// TIA Portal V16 export
// export: Created 2023-03-29T11:04:38.4378886Z, ExportSetting WithDefaults, DisplayName Totally Integrated Automation Portal, DisplayVersion V16 Update 6, DisplayName TIA Portal Version Control Interface, DisplayVersion V16 Update 2, DisplayName TIA Portal Openness, DisplayVersion V16 Update 6, DisplayName STEP 7 Professional, DisplayVersion V16 Update 6, DisplayName STEP 7 Safety, DisplayVersion V16, DisplayName WinCC Advanced, DisplayVersion V16 Update 6
FUNCTION "MPP04_2_rez" : Void   // FC24, LAD
TITLE = Read data from SC100
{ S7_Optimized_Access := 'TRUE' }
AUTHOR : rtecmer
VERSION : 0.1
// Czytanie z SC1000 
// Obsługa protokołu Master Modbus RTU.  Odczyt pomiarów  i status czujnika SC1000
// stored: AutoNumber false, IsIECCheckEnabled false, SetENOAutomatically false, UDAEnableTagReadback false
   VAR_TEMP
      Wielkość_przeływu_Adres0_0 : DWord;
      Wielkość_przeływu_Adres0_1 : DWord;
      Wielkość_przeływu_Adres2_0 : DWord;
      Wielkość_przeływu_Adres2_2 : DWord;
   END_VAR
   VAR_TEMP   // added for the SCL form of the ladder/FBD networks
      _w1 : Bool;
      _w2 : Bool;
   END_VAR
BEGIN

REGION Network 1
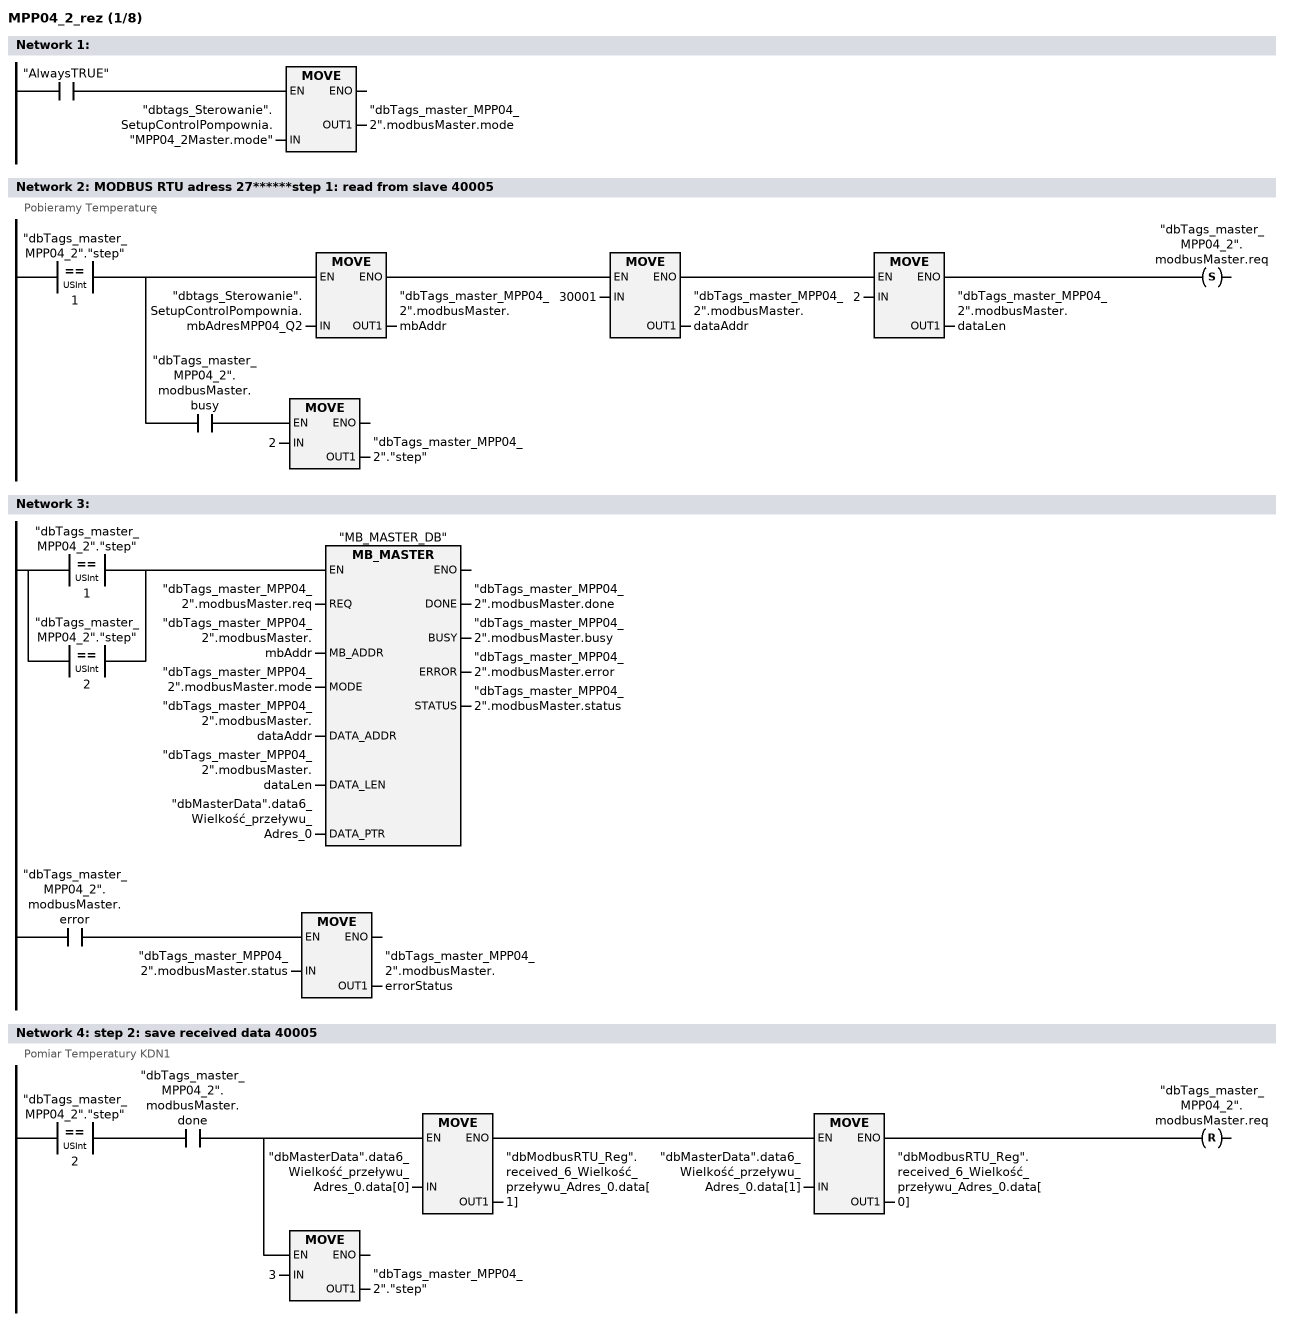
   RUNG wire#powerrail
      Contact( "AlwaysTRUE" )
      { S7_GenerateENO := "TRUE" } Move(in := "dbtags_Sterowanie".SetupControlPompownia."MPP04_2Master.mode", out1 => "dbTags_master_MPP04_2".modbusMaster.mode)
   END_RUNG
   // the same network as SCL:
   IF "AlwaysTRUE" THEN
       "dbTags_master_MPP04_2".modbusMaster.mode := "dbtags_Sterowanie".SetupControlPompownia."MPP04_2Master.mode";
   END_IF;
END_REGION

REGION Network 2: MODBUS RTU adress 27******step 1: read from slave 40005
   // Pobieramy Temperaturę
   RUNG wire#powerrail
      { S7_Templates := "SrcType := USInt" } EQ_Contact(in1 := "dbTags_master_MPP04_2"."step", in2 := 1)
      wire#w1
      Move(in := "dbtags_Sterowanie".SetupControlPompownia.mbAdresMPP04_Q2, out1 => "dbTags_master_MPP04_2".modbusMaster.mbAddr)
      { S7_GenerateENO := "TRUE" } Move(in := 30001, out1 => "dbTags_master_MPP04_2".modbusMaster.dataAddr)
      Move(in := 2, out1 => "dbTags_master_MPP04_2".modbusMaster.dataLen)
      S_Coil( "dbTags_master_MPP04_2".modbusMaster.req )
   END_RUNG
   RUNG wire#w1
      Contact( "dbTags_master_MPP04_2".modbusMaster.busy )
      { S7_GenerateENO := "TRUE" } Move(in := 2, out1 => "dbTags_master_MPP04_2"."step")
   END_RUNG
   // the same network as SCL:
   // ENO of a box is taken as its EN; it also drops when the box reports an error
   #_w1 := "dbTags_master_MPP04_2"."step" = 1;
   IF #_w1 THEN
       "dbTags_master_MPP04_2".modbusMaster.mbAddr := "dbtags_Sterowanie".SetupControlPompownia.mbAdresMPP04_Q2;
       "dbTags_master_MPP04_2".modbusMaster.dataAddr := 30001;
       "dbTags_master_MPP04_2".modbusMaster.dataLen := 2;
       "dbTags_master_MPP04_2".modbusMaster.req := TRUE;
   END_IF;
   IF #_w1 AND "dbTags_master_MPP04_2".modbusMaster.busy THEN "dbTags_master_MPP04_2"."step" := 2; END_IF;
END_REGION

REGION Network 3
   RUNG wire#powerrail
      { S7_Templates := "SrcType := USInt" } EQ_Contact(in1 := "dbTags_master_MPP04_2"."step", in2 := 1)
      wire#w1
      "MB_MASTER_DB".MB_MASTER(REQ := "dbTags_master_MPP04_2".modbusMaster.req, MB_ADDR := "dbTags_master_MPP04_2".modbusMaster.mbAddr, MODE := "dbTags_master_MPP04_2".modbusMaster.mode, DATA_ADDR := "dbTags_master_MPP04_2".modbusMaster.dataAddr, DATA_LEN := "dbTags_master_MPP04_2".modbusMaster.dataLen, DATA_PTR := "dbMasterData".data6_Wielkość_przeływu_Adres_0, DONE => "dbTags_master_MPP04_2".modbusMaster.done, BUSY => "dbTags_master_MPP04_2".modbusMaster.busy, ERROR => "dbTags_master_MPP04_2".modbusMaster.error, STATUS => "dbTags_master_MPP04_2".modbusMaster.status)
   END_RUNG
   RUNG wire#powerrail
      { S7_Templates := "SrcType := USInt" } EQ_Contact(in1 := "dbTags_master_MPP04_2"."step", in2 := 2)
   END_RUNG wire#w1
   RUNG wire#powerrail
      Contact( "dbTags_master_MPP04_2".modbusMaster.error )
      { S7_GenerateENO := "TRUE" } Move(in := "dbTags_master_MPP04_2".modbusMaster.status, out1 => "dbTags_master_MPP04_2".modbusMaster.errorStatus)
   END_RUNG
   // the same network as SCL:
   IF ("dbTags_master_MPP04_2"."step" = 1) OR ("dbTags_master_MPP04_2"."step" = 2) THEN
       "MB_MASTER_DB"(REQ := "dbTags_master_MPP04_2".modbusMaster.req,   // MB_MASTER
                      MB_ADDR := "dbTags_master_MPP04_2".modbusMaster.mbAddr,
                      MODE := "dbTags_master_MPP04_2".modbusMaster.mode,
                      DATA_ADDR := "dbTags_master_MPP04_2".modbusMaster.dataAddr,
                      DATA_LEN := "dbTags_master_MPP04_2".modbusMaster.dataLen,
                      DATA_PTR := "dbMasterData".data6_Wielkość_przeływu_Adres_0,
                      DONE => "dbTags_master_MPP04_2".modbusMaster.done,
                      BUSY => "dbTags_master_MPP04_2".modbusMaster.busy,
                      ERROR => "dbTags_master_MPP04_2".modbusMaster.error,
                      STATUS => "dbTags_master_MPP04_2".modbusMaster.status);
   END_IF;
   IF "dbTags_master_MPP04_2".modbusMaster.error THEN
       "dbTags_master_MPP04_2".modbusMaster.errorStatus := "dbTags_master_MPP04_2".modbusMaster.status;
   END_IF;
END_REGION

REGION Network 4: step 2: save received data 40005
   // Pomiar Temperatury KDN1
   RUNG wire#powerrail
      { S7_Templates := "SrcType := USInt" } EQ_Contact(in1 := "dbTags_master_MPP04_2"."step", in2 := 2)
      Contact( "dbTags_master_MPP04_2".modbusMaster.done )
      wire#w1
      { S7_GenerateENO := "TRUE" } Move(in := "dbMasterData".data6_Wielkość_przeływu_Adres_0.data[0], out1 => "dbModbusRTU_Reg".received_6_Wielkość_przeływu_Adres_0.data[1])
      { S7_GenerateENO := "TRUE" } Move(in := "dbMasterData".data6_Wielkość_przeływu_Adres_0.data[1], out1 => "dbModbusRTU_Reg".received_6_Wielkość_przeływu_Adres_0.data[0])
      R_Coil( "dbTags_master_MPP04_2".modbusMaster.req )
   END_RUNG
   RUNG wire#w1
      { S7_GenerateENO := "TRUE" } Move(in := 3, out1 => "dbTags_master_MPP04_2"."step")
   END_RUNG
   // the same network as SCL:
   // ENO of a box is taken as its EN; it also drops when the box reports an error
   IF ("dbTags_master_MPP04_2"."step" = 2) AND "dbTags_master_MPP04_2".modbusMaster.done THEN
       "dbModbusRTU_Reg".received_6_Wielkość_przeływu_Adres_0.data[1] := "dbMasterData".data6_Wielkość_przeływu_Adres_0.data[0];
       "dbModbusRTU_Reg".received_6_Wielkość_przeływu_Adres_0.data[0] := "dbMasterData".data6_Wielkość_przeływu_Adres_0.data[1];
       "dbTags_master_MPP04_2".modbusMaster.req := FALSE;
       "dbTags_master_MPP04_2"."step" := 3;
   END_IF;
END_REGION

REGION Network 5: MODBUS RTU adress 27******step 3: read from slave 40001
   // Bytes Error
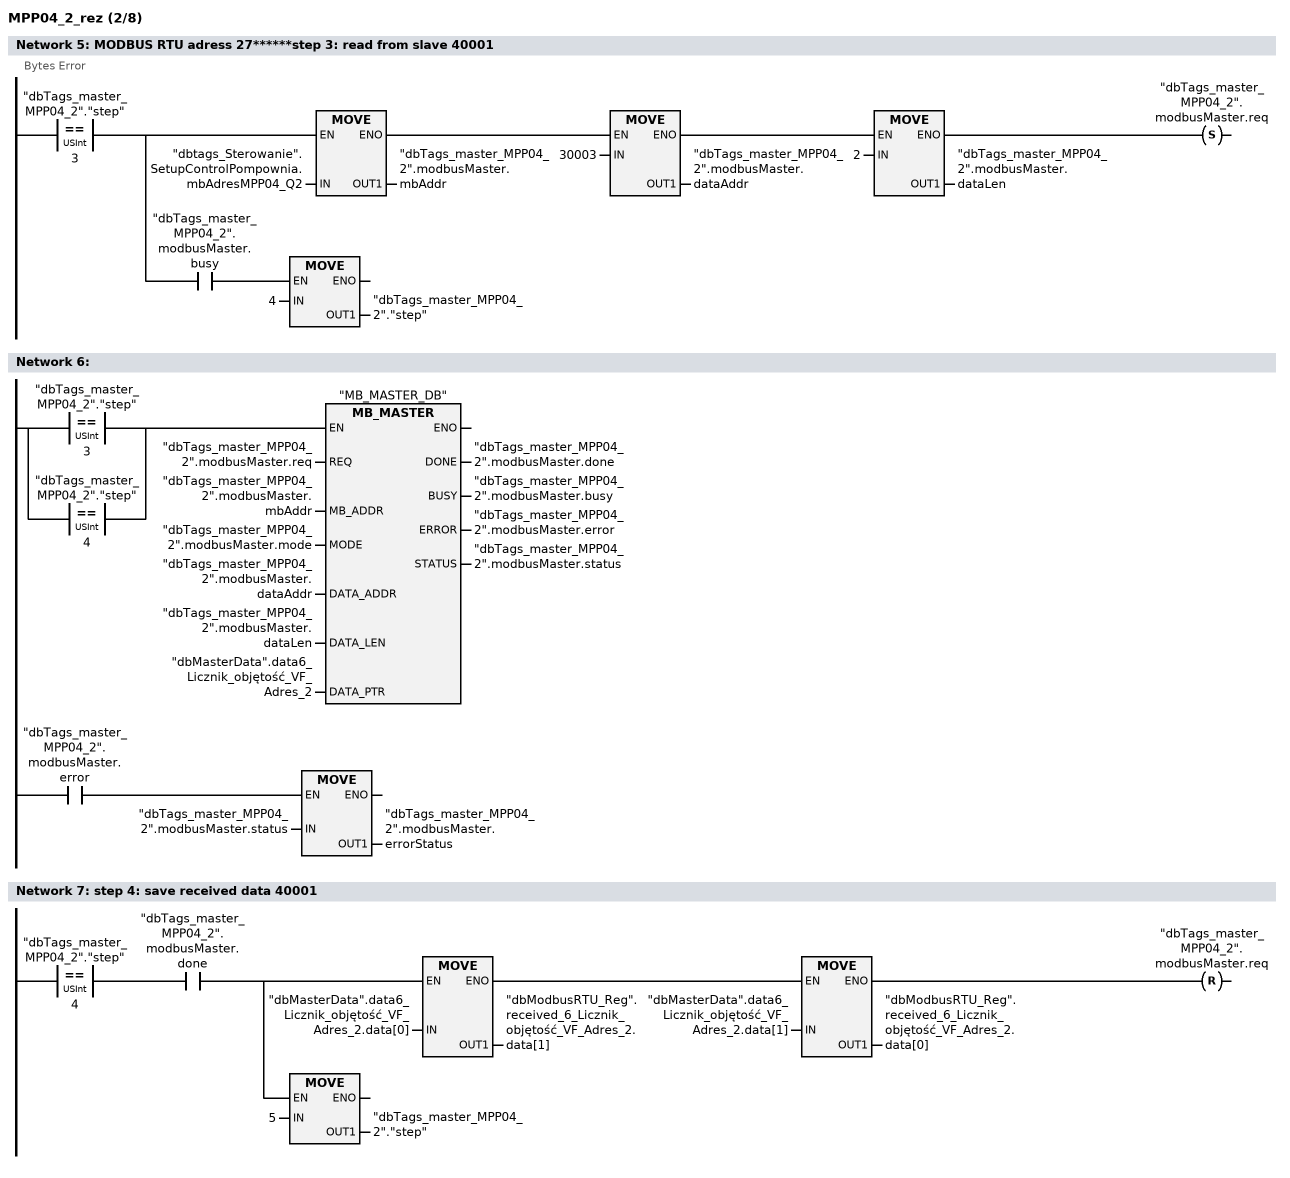
   RUNG wire#powerrail
      { S7_Templates := "SrcType := USInt" } EQ_Contact(in1 := "dbTags_master_MPP04_2"."step", in2 := 3)
      wire#w1
      Move(in := "dbtags_Sterowanie".SetupControlPompownia.mbAdresMPP04_Q2, out1 => "dbTags_master_MPP04_2".modbusMaster.mbAddr)
      { S7_GenerateENO := "TRUE" } Move(in := 30003, out1 => "dbTags_master_MPP04_2".modbusMaster.dataAddr)
      Move(in := 2, out1 => "dbTags_master_MPP04_2".modbusMaster.dataLen)
      S_Coil( "dbTags_master_MPP04_2".modbusMaster.req )
   END_RUNG
   RUNG wire#w1
      Contact( "dbTags_master_MPP04_2".modbusMaster.busy )
      { S7_GenerateENO := "TRUE" } Move(in := 4, out1 => "dbTags_master_MPP04_2"."step")
   END_RUNG
   // the same network as SCL:
   // ENO of a box is taken as its EN; it also drops when the box reports an error
   #_w1 := "dbTags_master_MPP04_2"."step" = 3;
   IF #_w1 THEN
       "dbTags_master_MPP04_2".modbusMaster.mbAddr := "dbtags_Sterowanie".SetupControlPompownia.mbAdresMPP04_Q2;
       "dbTags_master_MPP04_2".modbusMaster.dataAddr := 30003;
       "dbTags_master_MPP04_2".modbusMaster.dataLen := 2;
       "dbTags_master_MPP04_2".modbusMaster.req := TRUE;
   END_IF;
   IF #_w1 AND "dbTags_master_MPP04_2".modbusMaster.busy THEN "dbTags_master_MPP04_2"."step" := 4; END_IF;
END_REGION

REGION Network 6
   RUNG wire#powerrail
      { S7_Templates := "SrcType := USInt" } EQ_Contact(in1 := "dbTags_master_MPP04_2"."step", in2 := 3)
      wire#w1
      "MB_MASTER_DB".MB_MASTER(REQ := "dbTags_master_MPP04_2".modbusMaster.req, MB_ADDR := "dbTags_master_MPP04_2".modbusMaster.mbAddr, MODE := "dbTags_master_MPP04_2".modbusMaster.mode, DATA_ADDR := "dbTags_master_MPP04_2".modbusMaster.dataAddr, DATA_LEN := "dbTags_master_MPP04_2".modbusMaster.dataLen, DATA_PTR := "dbMasterData".data6_Licznik_objętość_VF_Adres_2, DONE => "dbTags_master_MPP04_2".modbusMaster.done, BUSY => "dbTags_master_MPP04_2".modbusMaster.busy, ERROR => "dbTags_master_MPP04_2".modbusMaster.error, STATUS => "dbTags_master_MPP04_2".modbusMaster.status)
   END_RUNG
   RUNG wire#powerrail
      { S7_Templates := "SrcType := USInt" } EQ_Contact(in1 := "dbTags_master_MPP04_2"."step", in2 := 4)
   END_RUNG wire#w1
   RUNG wire#powerrail
      Contact( "dbTags_master_MPP04_2".modbusMaster.error )
      { S7_GenerateENO := "TRUE" } Move(in := "dbTags_master_MPP04_2".modbusMaster.status, out1 => "dbTags_master_MPP04_2".modbusMaster.errorStatus)
   END_RUNG
   // the same network as SCL:
   IF ("dbTags_master_MPP04_2"."step" = 3) OR ("dbTags_master_MPP04_2"."step" = 4) THEN
       "MB_MASTER_DB"(REQ := "dbTags_master_MPP04_2".modbusMaster.req,   // MB_MASTER
                      MB_ADDR := "dbTags_master_MPP04_2".modbusMaster.mbAddr,
                      MODE := "dbTags_master_MPP04_2".modbusMaster.mode,
                      DATA_ADDR := "dbTags_master_MPP04_2".modbusMaster.dataAddr,
                      DATA_LEN := "dbTags_master_MPP04_2".modbusMaster.dataLen,
                      DATA_PTR := "dbMasterData".data6_Licznik_objętość_VF_Adres_2,
                      DONE => "dbTags_master_MPP04_2".modbusMaster.done,
                      BUSY => "dbTags_master_MPP04_2".modbusMaster.busy,
                      ERROR => "dbTags_master_MPP04_2".modbusMaster.error,
                      STATUS => "dbTags_master_MPP04_2".modbusMaster.status);
   END_IF;
   IF "dbTags_master_MPP04_2".modbusMaster.error THEN
       "dbTags_master_MPP04_2".modbusMaster.errorStatus := "dbTags_master_MPP04_2".modbusMaster.status;
   END_IF;
END_REGION

REGION Network 7: step 4: save received data 40001
   RUNG wire#powerrail
      { S7_Templates := "SrcType := USInt" } EQ_Contact(in1 := "dbTags_master_MPP04_2"."step", in2 := 4)
      Contact( "dbTags_master_MPP04_2".modbusMaster.done )
      wire#w1
      { S7_GenerateENO := "TRUE" } Move(in := "dbMasterData".data6_Licznik_objętość_VF_Adres_2.data[0], out1 => "dbModbusRTU_Reg".received_6_Licznik_objętość_VF_Adres_2.data[1])
      { S7_GenerateENO := "TRUE" } Move(in := "dbMasterData".data6_Licznik_objętość_VF_Adres_2.data[1], out1 => "dbModbusRTU_Reg".received_6_Licznik_objętość_VF_Adres_2.data[0])
      R_Coil( "dbTags_master_MPP04_2".modbusMaster.req )
   END_RUNG
   RUNG wire#w1
      { S7_GenerateENO := "TRUE" } Move(in := 5, out1 => "dbTags_master_MPP04_2"."step")
   END_RUNG
   // the same network as SCL:
   // ENO of a box is taken as its EN; it also drops when the box reports an error
   IF ("dbTags_master_MPP04_2"."step" = 4) AND "dbTags_master_MPP04_2".modbusMaster.done THEN
       "dbModbusRTU_Reg".received_6_Licznik_objętość_VF_Adres_2.data[1] := "dbMasterData".data6_Licznik_objętość_VF_Adres_2.data[0];
       "dbModbusRTU_Reg".received_6_Licznik_objętość_VF_Adres_2.data[0] := "dbMasterData".data6_Licznik_objętość_VF_Adres_2.data[1];
       "dbTags_master_MPP04_2".modbusMaster.req := FALSE;
       "dbTags_master_MPP04_2"."step" := 5;
   END_IF;
END_REGION

REGION Network 8: MODBUS RTU adress 27******step 5: read from slave 40002
   // Pobieramy status sondy
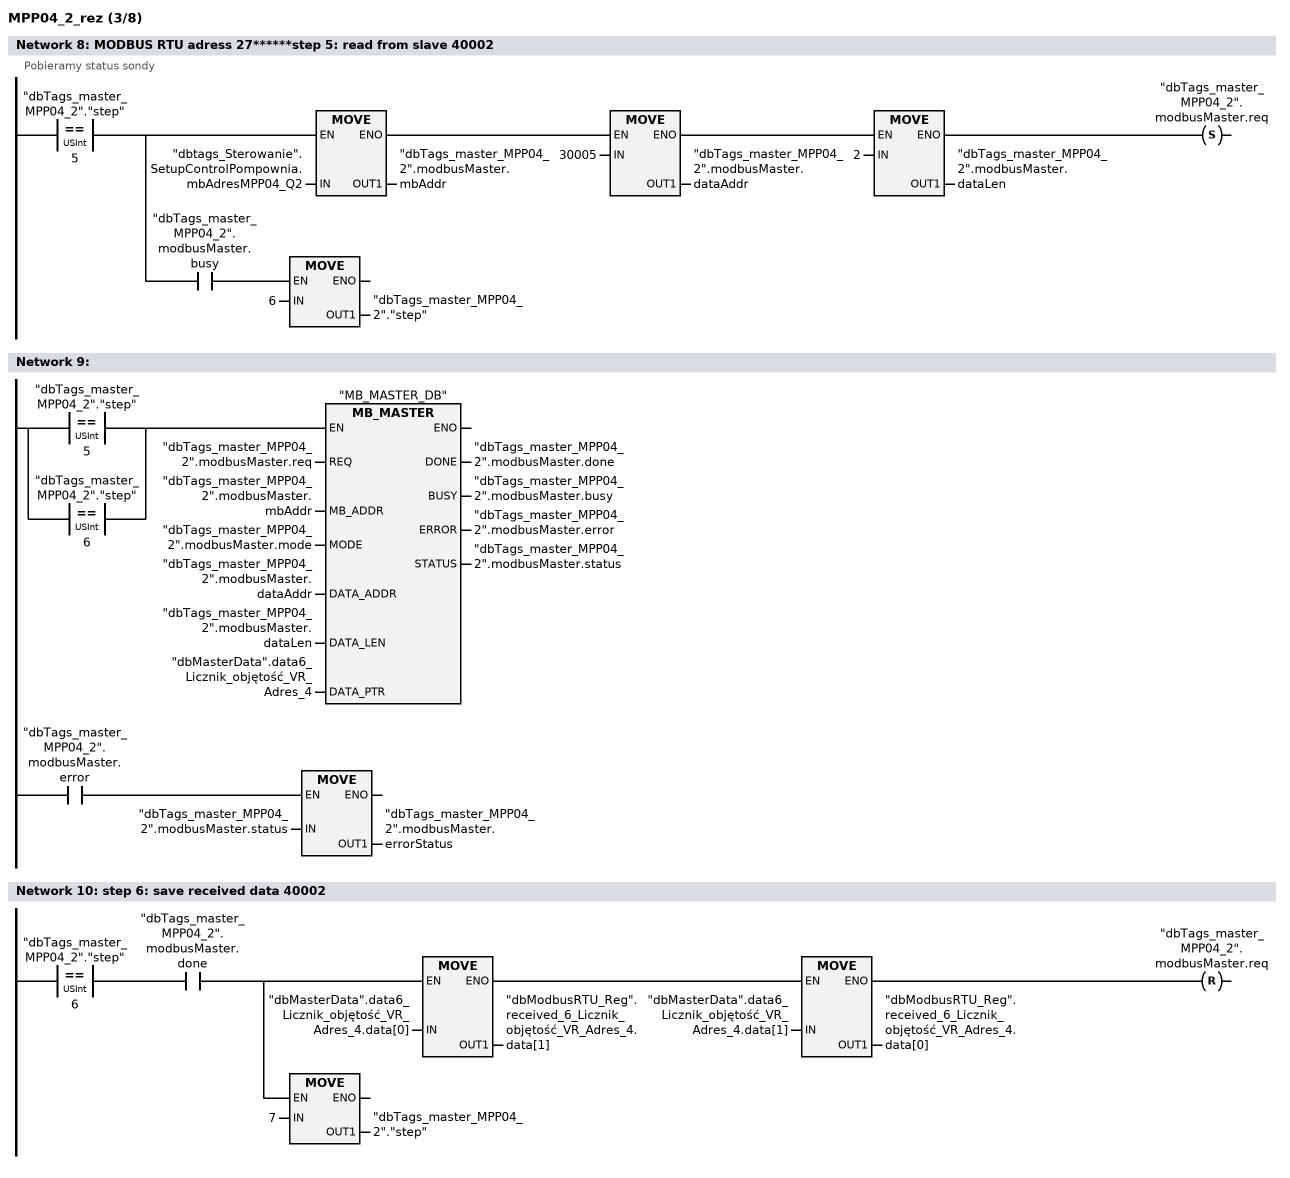
   RUNG wire#powerrail
      { S7_Templates := "SrcType := USInt" } EQ_Contact(in1 := "dbTags_master_MPP04_2"."step", in2 := 5)
      wire#w1
      Move(in := "dbtags_Sterowanie".SetupControlPompownia.mbAdresMPP04_Q2, out1 => "dbTags_master_MPP04_2".modbusMaster.mbAddr)
      { S7_GenerateENO := "TRUE" } Move(in := 30005, out1 => "dbTags_master_MPP04_2".modbusMaster.dataAddr)
      Move(in := 2, out1 => "dbTags_master_MPP04_2".modbusMaster.dataLen)
      S_Coil( "dbTags_master_MPP04_2".modbusMaster.req )
   END_RUNG
   RUNG wire#w1
      Contact( "dbTags_master_MPP04_2".modbusMaster.busy )
      { S7_GenerateENO := "TRUE" } Move(in := 6, out1 => "dbTags_master_MPP04_2"."step")
   END_RUNG
   // the same network as SCL:
   // ENO of a box is taken as its EN; it also drops when the box reports an error
   #_w1 := "dbTags_master_MPP04_2"."step" = 5;
   IF #_w1 THEN
       "dbTags_master_MPP04_2".modbusMaster.mbAddr := "dbtags_Sterowanie".SetupControlPompownia.mbAdresMPP04_Q2;
       "dbTags_master_MPP04_2".modbusMaster.dataAddr := 30005;
       "dbTags_master_MPP04_2".modbusMaster.dataLen := 2;
       "dbTags_master_MPP04_2".modbusMaster.req := TRUE;
   END_IF;
   IF #_w1 AND "dbTags_master_MPP04_2".modbusMaster.busy THEN "dbTags_master_MPP04_2"."step" := 6; END_IF;
END_REGION

REGION Network 9
   RUNG wire#powerrail
      { S7_Templates := "SrcType := USInt" } EQ_Contact(in1 := "dbTags_master_MPP04_2"."step", in2 := 5)
      wire#w1
      "MB_MASTER_DB".MB_MASTER(REQ := "dbTags_master_MPP04_2".modbusMaster.req, MB_ADDR := "dbTags_master_MPP04_2".modbusMaster.mbAddr, MODE := "dbTags_master_MPP04_2".modbusMaster.mode, DATA_ADDR := "dbTags_master_MPP04_2".modbusMaster.dataAddr, DATA_LEN := "dbTags_master_MPP04_2".modbusMaster.dataLen, DATA_PTR := "dbMasterData".data6_Licznik_objętość_VR_Adres_4, DONE => "dbTags_master_MPP04_2".modbusMaster.done, BUSY => "dbTags_master_MPP04_2".modbusMaster.busy, ERROR => "dbTags_master_MPP04_2".modbusMaster.error, STATUS => "dbTags_master_MPP04_2".modbusMaster.status)
   END_RUNG
   RUNG wire#powerrail
      { S7_Templates := "SrcType := USInt" } EQ_Contact(in1 := "dbTags_master_MPP04_2"."step", in2 := 6)
   END_RUNG wire#w1
   RUNG wire#powerrail
      Contact( "dbTags_master_MPP04_2".modbusMaster.error )
      { S7_GenerateENO := "TRUE" } Move(in := "dbTags_master_MPP04_2".modbusMaster.status, out1 => "dbTags_master_MPP04_2".modbusMaster.errorStatus)
   END_RUNG
   // the same network as SCL:
   IF ("dbTags_master_MPP04_2"."step" = 5) OR ("dbTags_master_MPP04_2"."step" = 6) THEN
       "MB_MASTER_DB"(REQ := "dbTags_master_MPP04_2".modbusMaster.req,   // MB_MASTER
                      MB_ADDR := "dbTags_master_MPP04_2".modbusMaster.mbAddr,
                      MODE := "dbTags_master_MPP04_2".modbusMaster.mode,
                      DATA_ADDR := "dbTags_master_MPP04_2".modbusMaster.dataAddr,
                      DATA_LEN := "dbTags_master_MPP04_2".modbusMaster.dataLen,
                      DATA_PTR := "dbMasterData".data6_Licznik_objętość_VR_Adres_4,
                      DONE => "dbTags_master_MPP04_2".modbusMaster.done,
                      BUSY => "dbTags_master_MPP04_2".modbusMaster.busy,
                      ERROR => "dbTags_master_MPP04_2".modbusMaster.error,
                      STATUS => "dbTags_master_MPP04_2".modbusMaster.status);
   END_IF;
   IF "dbTags_master_MPP04_2".modbusMaster.error THEN
       "dbTags_master_MPP04_2".modbusMaster.errorStatus := "dbTags_master_MPP04_2".modbusMaster.status;
   END_IF;
END_REGION

REGION Network 10: step 6: save received data 40002
   RUNG wire#powerrail
      { S7_Templates := "SrcType := USInt" } EQ_Contact(in1 := "dbTags_master_MPP04_2"."step", in2 := 6)
      Contact( "dbTags_master_MPP04_2".modbusMaster.done )
      wire#w1
      { S7_GenerateENO := "TRUE" } Move(in := "dbMasterData".data6_Licznik_objętość_VR_Adres_4.data[0], out1 => "dbModbusRTU_Reg".received_6_Licznik_objętość_VR_Adres_4.data[1])
      { S7_GenerateENO := "TRUE" } Move(in := "dbMasterData".data6_Licznik_objętość_VR_Adres_4.data[1], out1 => "dbModbusRTU_Reg".received_6_Licznik_objętość_VR_Adres_4.data[0])
      R_Coil( "dbTags_master_MPP04_2".modbusMaster.req )
   END_RUNG
   RUNG wire#w1
      { S7_GenerateENO := "TRUE" } Move(in := 7, out1 => "dbTags_master_MPP04_2"."step")
   END_RUNG
   // the same network as SCL:
   // ENO of a box is taken as its EN; it also drops when the box reports an error
   IF ("dbTags_master_MPP04_2"."step" = 6) AND "dbTags_master_MPP04_2".modbusMaster.done THEN
       "dbModbusRTU_Reg".received_6_Licznik_objętość_VR_Adres_4.data[1] := "dbMasterData".data6_Licznik_objętość_VR_Adres_4.data[0];
       "dbModbusRTU_Reg".received_6_Licznik_objętość_VR_Adres_4.data[0] := "dbMasterData".data6_Licznik_objętość_VR_Adres_4.data[1];
       "dbTags_master_MPP04_2".modbusMaster.req := FALSE;
       "dbTags_master_MPP04_2"."step" := 7;
   END_IF;
END_REGION

REGION Network 11: MODBUS RTU adress 27******step 9: read from slave 400011
   // Pobieramy Temperaturę w KN2
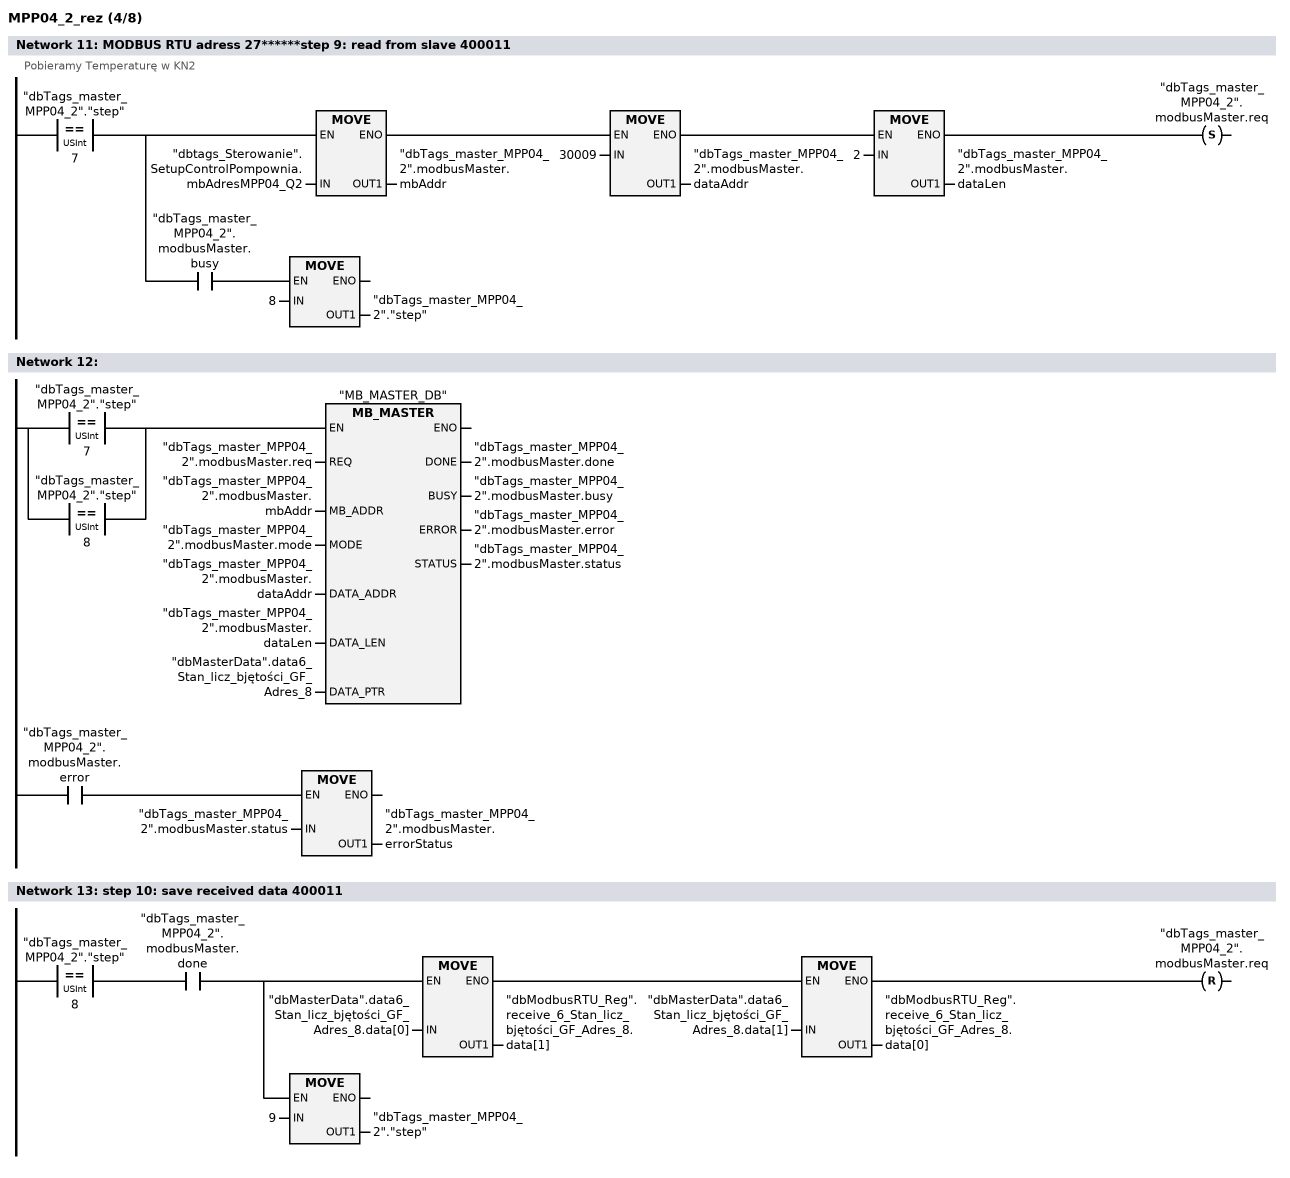
   RUNG wire#powerrail
      { S7_Templates := "SrcType := USInt" } EQ_Contact(in1 := "dbTags_master_MPP04_2"."step", in2 := 7)
      wire#w1
      Move(in := "dbtags_Sterowanie".SetupControlPompownia.mbAdresMPP04_Q2, out1 => "dbTags_master_MPP04_2".modbusMaster.mbAddr)
      { S7_GenerateENO := "TRUE" } Move(in := 30009, out1 => "dbTags_master_MPP04_2".modbusMaster.dataAddr)
      Move(in := 2, out1 => "dbTags_master_MPP04_2".modbusMaster.dataLen)
      S_Coil( "dbTags_master_MPP04_2".modbusMaster.req )
   END_RUNG
   RUNG wire#w1
      Contact( "dbTags_master_MPP04_2".modbusMaster.busy )
      { S7_GenerateENO := "TRUE" } Move(in := 8, out1 => "dbTags_master_MPP04_2"."step")
   END_RUNG
   // the same network as SCL:
   // ENO of a box is taken as its EN; it also drops when the box reports an error
   #_w1 := "dbTags_master_MPP04_2"."step" = 7;
   IF #_w1 THEN
       "dbTags_master_MPP04_2".modbusMaster.mbAddr := "dbtags_Sterowanie".SetupControlPompownia.mbAdresMPP04_Q2;
       "dbTags_master_MPP04_2".modbusMaster.dataAddr := 30009;
       "dbTags_master_MPP04_2".modbusMaster.dataLen := 2;
       "dbTags_master_MPP04_2".modbusMaster.req := TRUE;
   END_IF;
   IF #_w1 AND "dbTags_master_MPP04_2".modbusMaster.busy THEN "dbTags_master_MPP04_2"."step" := 8; END_IF;
END_REGION

REGION Network 12
   RUNG wire#powerrail
      { S7_Templates := "SrcType := USInt" } EQ_Contact(in1 := "dbTags_master_MPP04_2"."step", in2 := 7)
      wire#w1
      "MB_MASTER_DB".MB_MASTER(REQ := "dbTags_master_MPP04_2".modbusMaster.req, MB_ADDR := "dbTags_master_MPP04_2".modbusMaster.mbAddr, MODE := "dbTags_master_MPP04_2".modbusMaster.mode, DATA_ADDR := "dbTags_master_MPP04_2".modbusMaster.dataAddr, DATA_LEN := "dbTags_master_MPP04_2".modbusMaster.dataLen, DATA_PTR := "dbMasterData".data6_Stan_licz_bjętości_GF_Adres_8, DONE => "dbTags_master_MPP04_2".modbusMaster.done, BUSY => "dbTags_master_MPP04_2".modbusMaster.busy, ERROR => "dbTags_master_MPP04_2".modbusMaster.error, STATUS => "dbTags_master_MPP04_2".modbusMaster.status)
   END_RUNG
   RUNG wire#powerrail
      { S7_Templates := "SrcType := USInt" } EQ_Contact(in1 := "dbTags_master_MPP04_2"."step", in2 := 8)
   END_RUNG wire#w1
   RUNG wire#powerrail
      Contact( "dbTags_master_MPP04_2".modbusMaster.error )
      { S7_GenerateENO := "TRUE" } Move(in := "dbTags_master_MPP04_2".modbusMaster.status, out1 => "dbTags_master_MPP04_2".modbusMaster.errorStatus)
   END_RUNG
   // the same network as SCL:
   IF ("dbTags_master_MPP04_2"."step" = 7) OR ("dbTags_master_MPP04_2"."step" = 8) THEN
       "MB_MASTER_DB"(REQ := "dbTags_master_MPP04_2".modbusMaster.req,   // MB_MASTER
                      MB_ADDR := "dbTags_master_MPP04_2".modbusMaster.mbAddr,
                      MODE := "dbTags_master_MPP04_2".modbusMaster.mode,
                      DATA_ADDR := "dbTags_master_MPP04_2".modbusMaster.dataAddr,
                      DATA_LEN := "dbTags_master_MPP04_2".modbusMaster.dataLen,
                      DATA_PTR := "dbMasterData".data6_Stan_licz_bjętości_GF_Adres_8,
                      DONE => "dbTags_master_MPP04_2".modbusMaster.done,
                      BUSY => "dbTags_master_MPP04_2".modbusMaster.busy,
                      ERROR => "dbTags_master_MPP04_2".modbusMaster.error,
                      STATUS => "dbTags_master_MPP04_2".modbusMaster.status);
   END_IF;
   IF "dbTags_master_MPP04_2".modbusMaster.error THEN
       "dbTags_master_MPP04_2".modbusMaster.errorStatus := "dbTags_master_MPP04_2".modbusMaster.status;
   END_IF;
END_REGION

REGION Network 13: step 10: save received data 400011
   RUNG wire#powerrail
      { S7_Templates := "SrcType := USInt" } EQ_Contact(in1 := "dbTags_master_MPP04_2"."step", in2 := 8)
      Contact( "dbTags_master_MPP04_2".modbusMaster.done )
      wire#w1
      { S7_GenerateENO := "TRUE" } Move(in := "dbMasterData".data6_Stan_licz_bjętości_GF_Adres_8.data[0], out1 => "dbModbusRTU_Reg".receive_6_Stan_licz_bjętości_GF_Adres_8.data[1])
      { S7_GenerateENO := "TRUE" } Move(in := "dbMasterData".data6_Stan_licz_bjętości_GF_Adres_8.data[1], out1 => "dbModbusRTU_Reg".receive_6_Stan_licz_bjętości_GF_Adres_8.data[0])
      R_Coil( "dbTags_master_MPP04_2".modbusMaster.req )
   END_RUNG
   RUNG wire#w1
      { S7_GenerateENO := "TRUE" } Move(in := 9, out1 => "dbTags_master_MPP04_2"."step")
   END_RUNG
   // the same network as SCL:
   // ENO of a box is taken as its EN; it also drops when the box reports an error
   IF ("dbTags_master_MPP04_2"."step" = 8) AND "dbTags_master_MPP04_2".modbusMaster.done THEN
       "dbModbusRTU_Reg".receive_6_Stan_licz_bjętości_GF_Adres_8.data[1] := "dbMasterData".data6_Stan_licz_bjętości_GF_Adres_8.data[0];
       "dbModbusRTU_Reg".receive_6_Stan_licz_bjętości_GF_Adres_8.data[0] := "dbMasterData".data6_Stan_licz_bjętości_GF_Adres_8.data[1];
       "dbTags_master_MPP04_2".modbusMaster.req := FALSE;
       "dbTags_master_MPP04_2"."step" := 9;
   END_IF;
END_REGION

REGION Network 14: MODBUS RTU adress 27******step 11: read from slave 40007
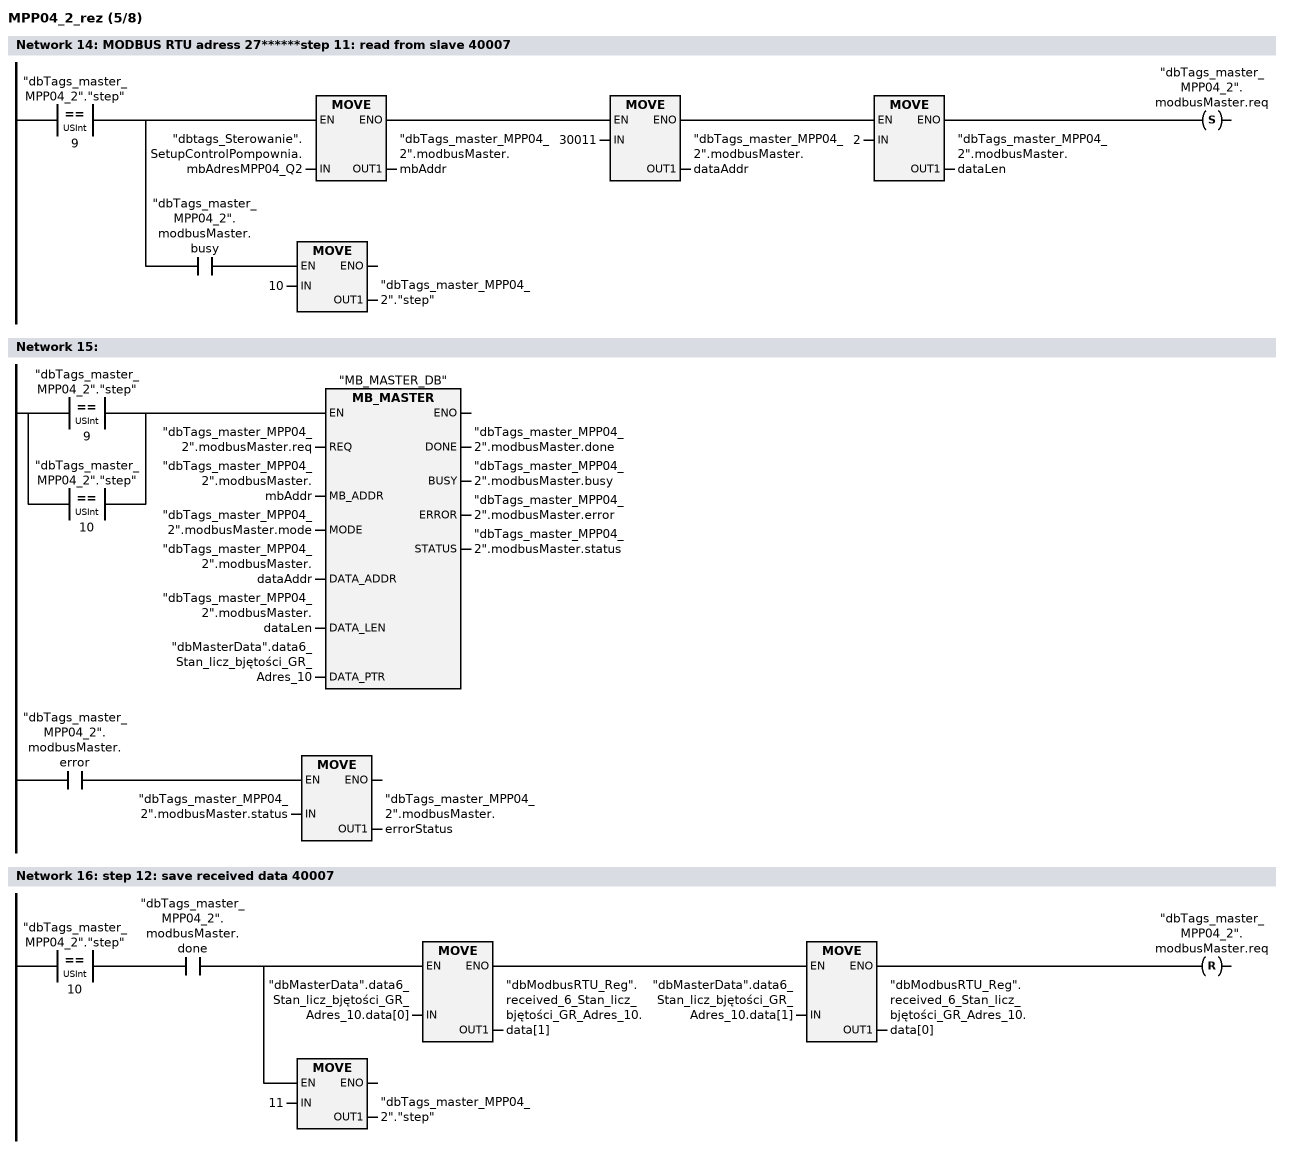
   RUNG wire#powerrail
      { S7_Templates := "SrcType := USInt" } EQ_Contact(in1 := "dbTags_master_MPP04_2"."step", in2 := 9)
      wire#w1
      Move(in := "dbtags_Sterowanie".SetupControlPompownia.mbAdresMPP04_Q2, out1 => "dbTags_master_MPP04_2".modbusMaster.mbAddr)
      { S7_GenerateENO := "TRUE" } Move(in := 30011, out1 => "dbTags_master_MPP04_2".modbusMaster.dataAddr)
      Move(in := 2, out1 => "dbTags_master_MPP04_2".modbusMaster.dataLen)
      S_Coil( "dbTags_master_MPP04_2".modbusMaster.req )
   END_RUNG
   RUNG wire#w1
      Contact( "dbTags_master_MPP04_2".modbusMaster.busy )
      { S7_GenerateENO := "TRUE" } Move(in := 10, out1 => "dbTags_master_MPP04_2"."step")
   END_RUNG
   // the same network as SCL:
   // ENO of a box is taken as its EN; it also drops when the box reports an error
   #_w1 := "dbTags_master_MPP04_2"."step" = 9;
   IF #_w1 THEN
       "dbTags_master_MPP04_2".modbusMaster.mbAddr := "dbtags_Sterowanie".SetupControlPompownia.mbAdresMPP04_Q2;
       "dbTags_master_MPP04_2".modbusMaster.dataAddr := 30011;
       "dbTags_master_MPP04_2".modbusMaster.dataLen := 2;
       "dbTags_master_MPP04_2".modbusMaster.req := TRUE;
   END_IF;
   IF #_w1 AND "dbTags_master_MPP04_2".modbusMaster.busy THEN "dbTags_master_MPP04_2"."step" := 10; END_IF;
END_REGION

REGION Network 15
   RUNG wire#powerrail
      { S7_Templates := "SrcType := USInt" } EQ_Contact(in1 := "dbTags_master_MPP04_2"."step", in2 := 9)
      wire#w1
      "MB_MASTER_DB".MB_MASTER(REQ := "dbTags_master_MPP04_2".modbusMaster.req, MB_ADDR := "dbTags_master_MPP04_2".modbusMaster.mbAddr, MODE := "dbTags_master_MPP04_2".modbusMaster.mode, DATA_ADDR := "dbTags_master_MPP04_2".modbusMaster.dataAddr, DATA_LEN := "dbTags_master_MPP04_2".modbusMaster.dataLen, DATA_PTR := "dbMasterData".data6_Stan_licz_bjętości_GR_Adres_10, DONE => "dbTags_master_MPP04_2".modbusMaster.done, BUSY => "dbTags_master_MPP04_2".modbusMaster.busy, ERROR => "dbTags_master_MPP04_2".modbusMaster.error, STATUS => "dbTags_master_MPP04_2".modbusMaster.status)
   END_RUNG
   RUNG wire#powerrail
      { S7_Templates := "SrcType := USInt" } EQ_Contact(in1 := "dbTags_master_MPP04_2"."step", in2 := 10)
   END_RUNG wire#w1
   RUNG wire#powerrail
      Contact( "dbTags_master_MPP04_2".modbusMaster.error )
      { S7_GenerateENO := "TRUE" } Move(in := "dbTags_master_MPP04_2".modbusMaster.status, out1 => "dbTags_master_MPP04_2".modbusMaster.errorStatus)
   END_RUNG
   // the same network as SCL:
   IF ("dbTags_master_MPP04_2"."step" = 9) OR ("dbTags_master_MPP04_2"."step" = 10) THEN
       "MB_MASTER_DB"(REQ := "dbTags_master_MPP04_2".modbusMaster.req,   // MB_MASTER
                      MB_ADDR := "dbTags_master_MPP04_2".modbusMaster.mbAddr,
                      MODE := "dbTags_master_MPP04_2".modbusMaster.mode,
                      DATA_ADDR := "dbTags_master_MPP04_2".modbusMaster.dataAddr,
                      DATA_LEN := "dbTags_master_MPP04_2".modbusMaster.dataLen,
                      DATA_PTR := "dbMasterData".data6_Stan_licz_bjętości_GR_Adres_10,
                      DONE => "dbTags_master_MPP04_2".modbusMaster.done,
                      BUSY => "dbTags_master_MPP04_2".modbusMaster.busy,
                      ERROR => "dbTags_master_MPP04_2".modbusMaster.error,
                      STATUS => "dbTags_master_MPP04_2".modbusMaster.status);
   END_IF;
   IF "dbTags_master_MPP04_2".modbusMaster.error THEN
       "dbTags_master_MPP04_2".modbusMaster.errorStatus := "dbTags_master_MPP04_2".modbusMaster.status;
   END_IF;
END_REGION

REGION Network 16: step 12: save received data 40007
   RUNG wire#powerrail
      { S7_Templates := "SrcType := USInt" } EQ_Contact(in1 := "dbTags_master_MPP04_2"."step", in2 := 10)
      Contact( "dbTags_master_MPP04_2".modbusMaster.done )
      wire#w1
      { S7_GenerateENO := "TRUE" } Move(in := "dbMasterData".data6_Stan_licz_bjętości_GR_Adres_10.data[0], out1 => "dbModbusRTU_Reg".received_6_Stan_licz_bjętości_GR_Adres_10.data[1])
      { S7_GenerateENO := "TRUE" } Move(in := "dbMasterData".data6_Stan_licz_bjętości_GR_Adres_10.data[1], out1 => "dbModbusRTU_Reg".received_6_Stan_licz_bjętości_GR_Adres_10.data[0])
      R_Coil( "dbTags_master_MPP04_2".modbusMaster.req )
   END_RUNG
   RUNG wire#w1
      { S7_GenerateENO := "TRUE" } Move(in := 11, out1 => "dbTags_master_MPP04_2"."step")
   END_RUNG
   // the same network as SCL:
   // ENO of a box is taken as its EN; it also drops when the box reports an error
   IF ("dbTags_master_MPP04_2"."step" = 10) AND "dbTags_master_MPP04_2".modbusMaster.done THEN
       "dbModbusRTU_Reg".received_6_Stan_licz_bjętości_GR_Adres_10.data[1] := "dbMasterData".data6_Stan_licz_bjętości_GR_Adres_10.data[0];
       "dbModbusRTU_Reg".received_6_Stan_licz_bjętości_GR_Adres_10.data[0] := "dbMasterData".data6_Stan_licz_bjętości_GR_Adres_10.data[1];
       "dbTags_master_MPP04_2".modbusMaster.req := FALSE;
       "dbTags_master_MPP04_2"."step" := 11;
   END_IF;
END_REGION

REGION Network 17: MODBUS RTU adress 27******step 15: read from slave 40009
   // Pobieramy  status urządzenia
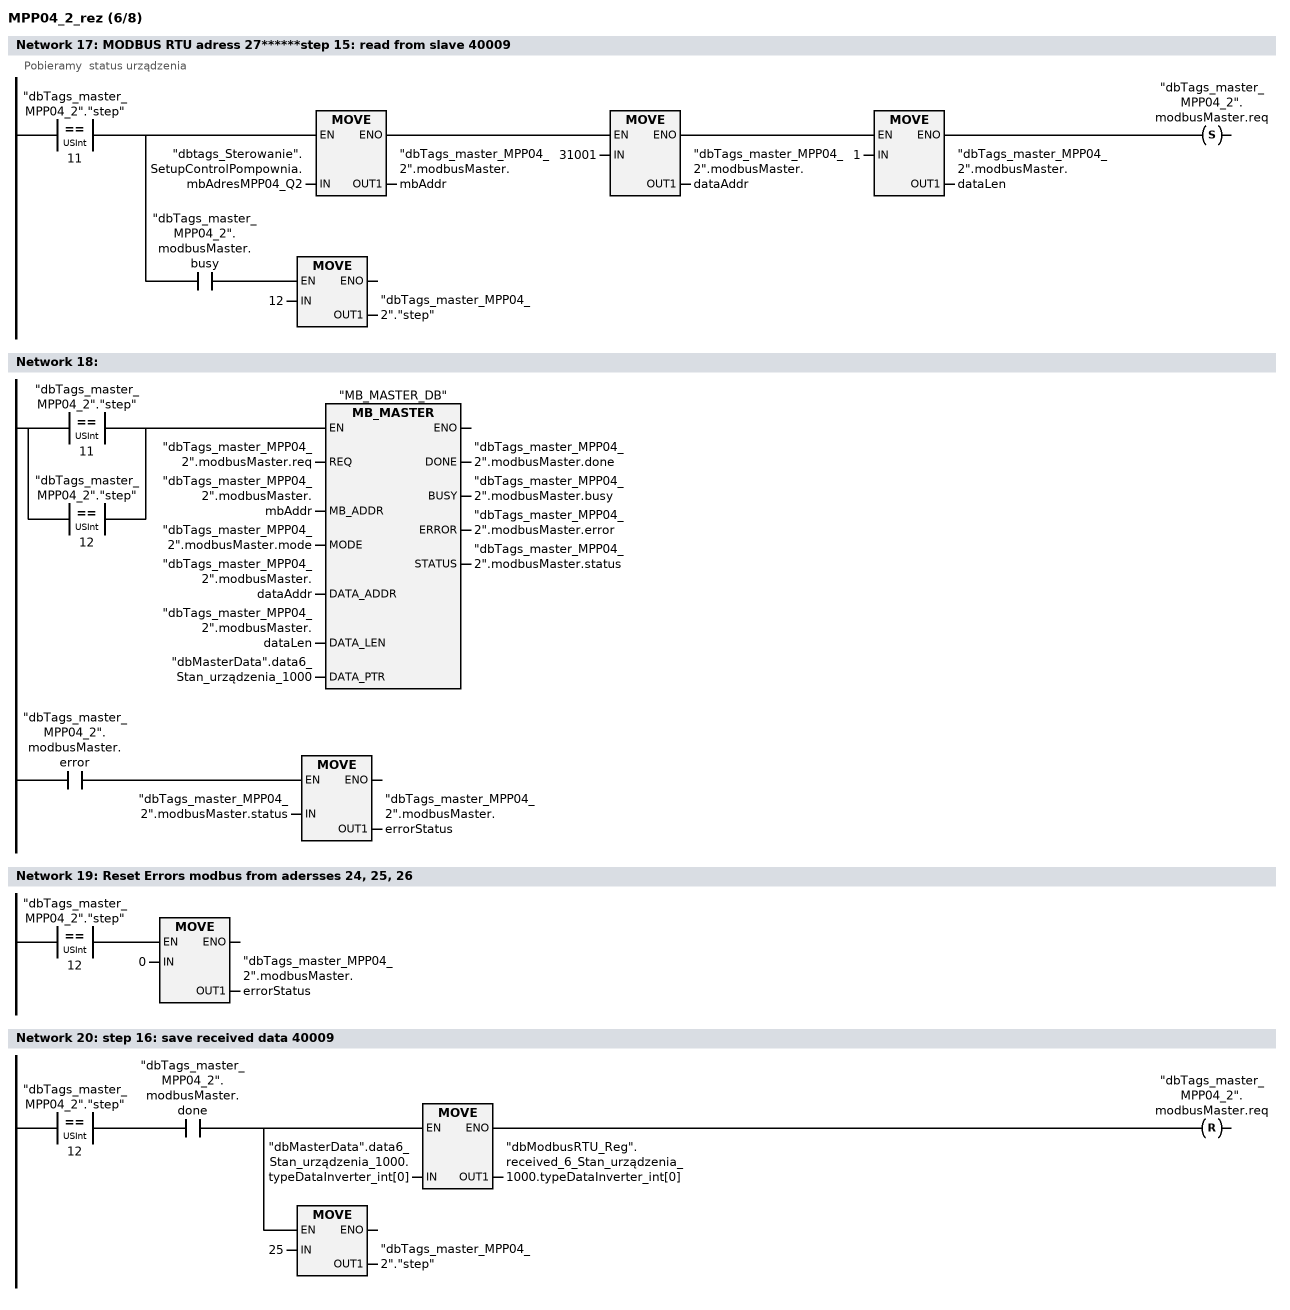
   RUNG wire#powerrail
      { S7_Templates := "SrcType := USInt" } EQ_Contact(in1 := "dbTags_master_MPP04_2"."step", in2 := 11)
      wire#w1
      Move(in := "dbtags_Sterowanie".SetupControlPompownia.mbAdresMPP04_Q2, out1 => "dbTags_master_MPP04_2".modbusMaster.mbAddr)
      { S7_GenerateENO := "TRUE" } Move(in := 31001, out1 => "dbTags_master_MPP04_2".modbusMaster.dataAddr)
      Move(in := 1, out1 => "dbTags_master_MPP04_2".modbusMaster.dataLen)
      S_Coil( "dbTags_master_MPP04_2".modbusMaster.req )
   END_RUNG
   RUNG wire#w1
      Contact( "dbTags_master_MPP04_2".modbusMaster.busy )
      { S7_GenerateENO := "TRUE" } Move(in := 12, out1 => "dbTags_master_MPP04_2"."step")
   END_RUNG
   // the same network as SCL:
   // ENO of a box is taken as its EN; it also drops when the box reports an error
   #_w1 := "dbTags_master_MPP04_2"."step" = 11;
   IF #_w1 THEN
       "dbTags_master_MPP04_2".modbusMaster.mbAddr := "dbtags_Sterowanie".SetupControlPompownia.mbAdresMPP04_Q2;
       "dbTags_master_MPP04_2".modbusMaster.dataAddr := 31001;
       "dbTags_master_MPP04_2".modbusMaster.dataLen := 1;
       "dbTags_master_MPP04_2".modbusMaster.req := TRUE;
   END_IF;
   IF #_w1 AND "dbTags_master_MPP04_2".modbusMaster.busy THEN "dbTags_master_MPP04_2"."step" := 12; END_IF;
END_REGION

REGION Network 18
   RUNG wire#powerrail
      { S7_Templates := "SrcType := USInt" } EQ_Contact(in1 := "dbTags_master_MPP04_2"."step", in2 := 11)
      wire#w1
      "MB_MASTER_DB".MB_MASTER(REQ := "dbTags_master_MPP04_2".modbusMaster.req, MB_ADDR := "dbTags_master_MPP04_2".modbusMaster.mbAddr, MODE := "dbTags_master_MPP04_2".modbusMaster.mode, DATA_ADDR := "dbTags_master_MPP04_2".modbusMaster.dataAddr, DATA_LEN := "dbTags_master_MPP04_2".modbusMaster.dataLen, DATA_PTR := "dbMasterData".data6_Stan_urządzenia_1000, DONE => "dbTags_master_MPP04_2".modbusMaster.done, BUSY => "dbTags_master_MPP04_2".modbusMaster.busy, ERROR => "dbTags_master_MPP04_2".modbusMaster.error, STATUS => "dbTags_master_MPP04_2".modbusMaster.status)
   END_RUNG
   RUNG wire#powerrail
      { S7_Templates := "SrcType := USInt" } EQ_Contact(in1 := "dbTags_master_MPP04_2"."step", in2 := 12)
   END_RUNG wire#w1
   RUNG wire#powerrail
      Contact( "dbTags_master_MPP04_2".modbusMaster.error )
      { S7_GenerateENO := "TRUE" } Move(in := "dbTags_master_MPP04_2".modbusMaster.status, out1 => "dbTags_master_MPP04_2".modbusMaster.errorStatus)
   END_RUNG
   // the same network as SCL:
   IF ("dbTags_master_MPP04_2"."step" = 11) OR ("dbTags_master_MPP04_2"."step" = 12) THEN
       "MB_MASTER_DB"(REQ := "dbTags_master_MPP04_2".modbusMaster.req,   // MB_MASTER
                      MB_ADDR := "dbTags_master_MPP04_2".modbusMaster.mbAddr,
                      MODE := "dbTags_master_MPP04_2".modbusMaster.mode,
                      DATA_ADDR := "dbTags_master_MPP04_2".modbusMaster.dataAddr,
                      DATA_LEN := "dbTags_master_MPP04_2".modbusMaster.dataLen,
                      DATA_PTR := "dbMasterData".data6_Stan_urządzenia_1000,
                      DONE => "dbTags_master_MPP04_2".modbusMaster.done,
                      BUSY => "dbTags_master_MPP04_2".modbusMaster.busy,
                      ERROR => "dbTags_master_MPP04_2".modbusMaster.error,
                      STATUS => "dbTags_master_MPP04_2".modbusMaster.status);
   END_IF;
   IF "dbTags_master_MPP04_2".modbusMaster.error THEN
       "dbTags_master_MPP04_2".modbusMaster.errorStatus := "dbTags_master_MPP04_2".modbusMaster.status;
   END_IF;
END_REGION

REGION Network 19: Reset Errors modbus from adersses 24, 25, 26
   RUNG wire#powerrail
      { S7_Templates := "SrcType := USInt" } EQ_Contact(in1 := "dbTags_master_MPP04_2"."step", in2 := 12)
      { S7_GenerateENO := "TRUE" } Move(in := 0, out1 => "dbTags_master_MPP04_2".modbusMaster.errorStatus)
   END_RUNG
   // the same network as SCL:
   IF "dbTags_master_MPP04_2"."step" = 12 THEN "dbTags_master_MPP04_2".modbusMaster.errorStatus := 0; END_IF;
END_REGION

REGION Network 20: step 16: save received data 40009
   RUNG wire#powerrail
      { S7_Templates := "SrcType := USInt" } EQ_Contact(in1 := "dbTags_master_MPP04_2"."step", in2 := 12)
      Contact( "dbTags_master_MPP04_2".modbusMaster.done )
      wire#w1
      { S7_GenerateENO := "TRUE" } Move(in := "dbMasterData".data6_Stan_urządzenia_1000.typeDataInverter_int[0], out1 => "dbModbusRTU_Reg".received_6_Stan_urządzenia_1000.typeDataInverter_int[0])
      R_Coil( "dbTags_master_MPP04_2".modbusMaster.req )
   END_RUNG
   RUNG wire#w1
      { S7_GenerateENO := "TRUE" } Move(in := 25, out1 => "dbTags_master_MPP04_2"."step")
   END_RUNG
   // the same network as SCL:
   // ENO of a box is taken as its EN; it also drops when the box reports an error
   IF ("dbTags_master_MPP04_2"."step" = 12) AND "dbTags_master_MPP04_2".modbusMaster.done THEN
       "dbModbusRTU_Reg".received_6_Stan_urządzenia_1000.typeDataInverter_int[0] := "dbMasterData".data6_Stan_urządzenia_1000.typeDataInverter_int[0];
       "dbTags_master_MPP04_2".modbusMaster.req := FALSE;
       "dbTags_master_MPP04_2"."step" := 25;
   END_IF;
END_REGION

REGION Network 21: Znacznik błedu komunikacji modbus
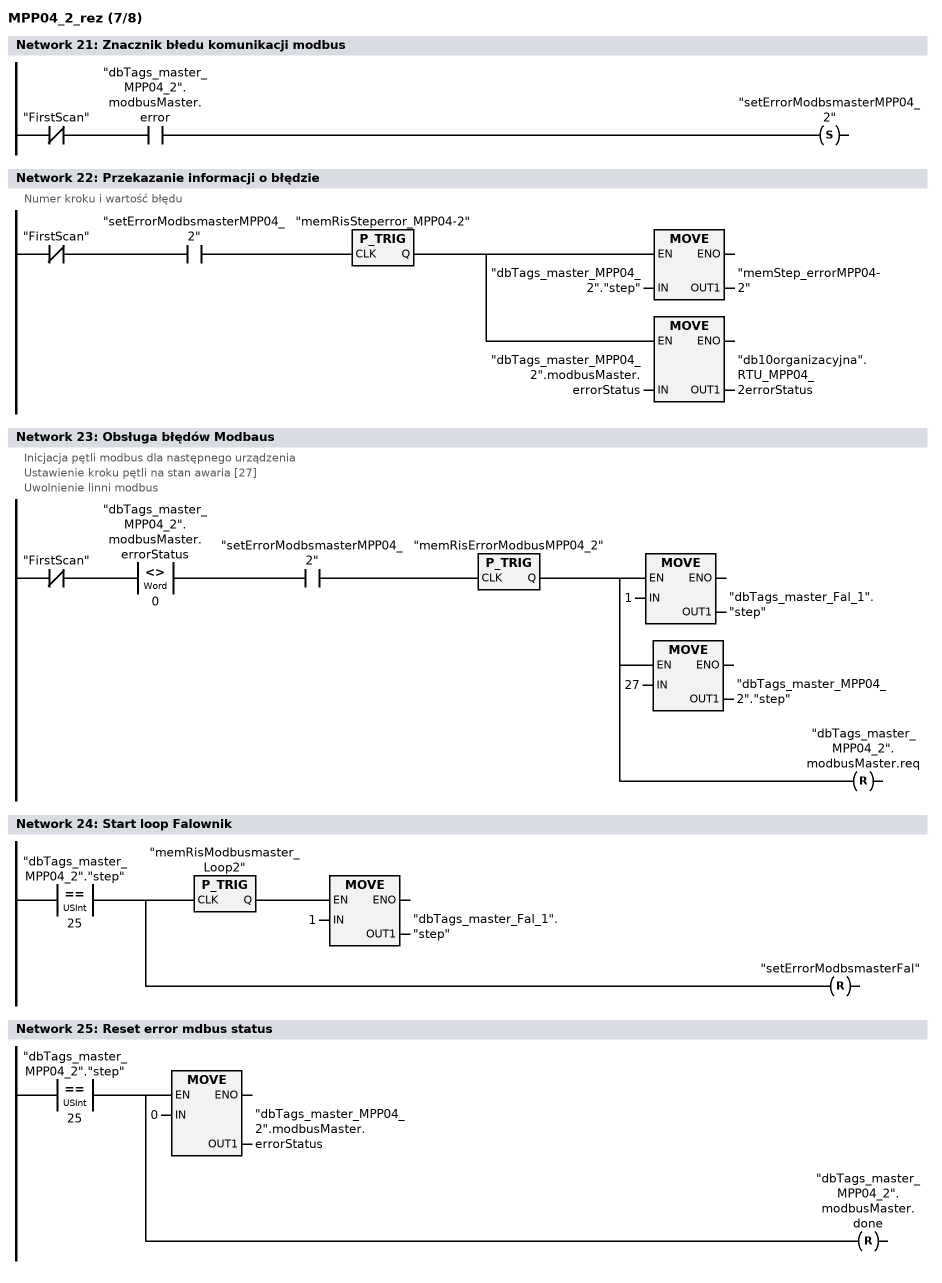
   RUNG wire#powerrail
      I_Contact( "FirstScan" )
      Contact( "dbTags_master_MPP04_2".modbusMaster.error )
      S_Coil( "setErrorModbsmasterMPP04_2" )
   END_RUNG
   // the same network as SCL:
   IF NOT "FirstScan" AND "dbTags_master_MPP04_2".modbusMaster.error THEN
       "setErrorModbsmasterMPP04_2" := TRUE;
   END_IF;
END_REGION

REGION Network 22: Przekazanie informacji o błędzie
   // Numer kroku i wartość błędu
   RUNG wire#powerrail
      I_Contact( "FirstScan" )
      Contact( "setErrorModbsmasterMPP04_2" )
      P_Trig( "memRisSteperror_MPP04-2" )
      wire#w1
      Move(in := "dbTags_master_MPP04_2"."step", out1 => "memStep_errorMPP04-2")
   END_RUNG
   RUNG wire#w1
      { S7_GenerateENO := "TRUE" } Move(in := "dbTags_master_MPP04_2".modbusMaster.errorStatus, out1 => "db10organizacyjna".RTU_MPP04_2errorStatus)
   END_RUNG
   // the same network as SCL:
   #_w1 := NOT "FirstScan" AND "setErrorModbsmasterMPP04_2";
   #_w2 := #_w1 AND NOT "memRisSteperror_MPP04-2";   // rising edge
   "memRisSteperror_MPP04-2" := #_w1;
   IF #_w2 THEN
       "memStep_errorMPP04-2" := "dbTags_master_MPP04_2"."step";
       "db10organizacyjna".RTU_MPP04_2errorStatus := "dbTags_master_MPP04_2".modbusMaster.errorStatus;
   END_IF;
END_REGION

REGION Network 23: Obsługa błędów Modbaus
   // Inicjacja pętli modbus dla następnego urządzenia
   // Ustawienie kroku pętli na stan awaria [27]
   // Uwolnienie linni modbus
   RUNG wire#powerrail
      I_Contact( "FirstScan" )
      { S7_Templates := "SrcType := Word" } NE_Contact(in1 := "dbTags_master_MPP04_2".modbusMaster.errorStatus, in2 := 0)
      Contact( "setErrorModbsmasterMPP04_2" )
      P_Trig( "memRisErrorModbusMPP04_2" )
      wire#w1
      { S7_GenerateENO := "TRUE" } Move(in := 1, out1 => "dbTags_master_Fal_1"."step")
   END_RUNG
   RUNG wire#w1
      { S7_GenerateENO := "TRUE" } Move(in := 27, out1 => "dbTags_master_MPP04_2"."step")
   END_RUNG
   RUNG wire#w1
      R_Coil( "dbTags_master_MPP04_2".modbusMaster.req )
   END_RUNG
   // the same network as SCL:
   #_w1 := NOT "FirstScan" AND ("dbTags_master_MPP04_2".modbusMaster.errorStatus <> 0) AND "setErrorModbsmasterMPP04_2";
   #_w2 := #_w1 AND NOT "memRisErrorModbusMPP04_2";   // rising edge
   "memRisErrorModbusMPP04_2" := #_w1;
   IF #_w2 THEN
       "dbTags_master_Fal_1"."step" := 1;
       "dbTags_master_MPP04_2"."step" := 27;
       "dbTags_master_MPP04_2".modbusMaster.req := FALSE;
   END_IF;
END_REGION

REGION Network 24: Start loop Falownik
   RUNG wire#powerrail
      { S7_Templates := "SrcType := USInt" } EQ_Contact(in1 := "dbTags_master_MPP04_2"."step", in2 := 25)
      wire#w1
      P_Trig( "memRisModbusmaster_Loop2" )
      { S7_GenerateENO := "TRUE" } Move(in := 1, out1 => "dbTags_master_Fal_1"."step")
   END_RUNG
   RUNG wire#w1
      R_Coil( "setErrorModbsmasterFal" )
   END_RUNG
   // the same network as SCL:
   #_w1 := "dbTags_master_MPP04_2"."step" = 25;
   #_w2 := #_w1 AND NOT "memRisModbusmaster_Loop2";   // rising edge
   "memRisModbusmaster_Loop2" := #_w1;
   IF #_w2 THEN "dbTags_master_Fal_1"."step" := 1; END_IF;
   IF #_w1 THEN "setErrorModbsmasterFal" := FALSE; END_IF;
END_REGION

REGION Network 25: Reset error mdbus status
   RUNG wire#powerrail
      { S7_Templates := "SrcType := USInt" } EQ_Contact(in1 := "dbTags_master_MPP04_2"."step", in2 := 25)
      wire#w1
      { S7_GenerateENO := "TRUE" } Move(in := 0, out1 => "dbTags_master_MPP04_2".modbusMaster.errorStatus)
   END_RUNG
   RUNG wire#w1
      R_Coil( "dbTags_master_MPP04_2".modbusMaster.done )
   END_RUNG
   // the same network as SCL:
   IF "dbTags_master_MPP04_2"."step" = 25 THEN
       "dbTags_master_MPP04_2".modbusMaster.errorStatus := 0;
       "dbTags_master_MPP04_2".modbusMaster.done := FALSE;
   END_IF;
END_REGION

REGION Network 26: Reset Znacznik błedu komunikacji modbus
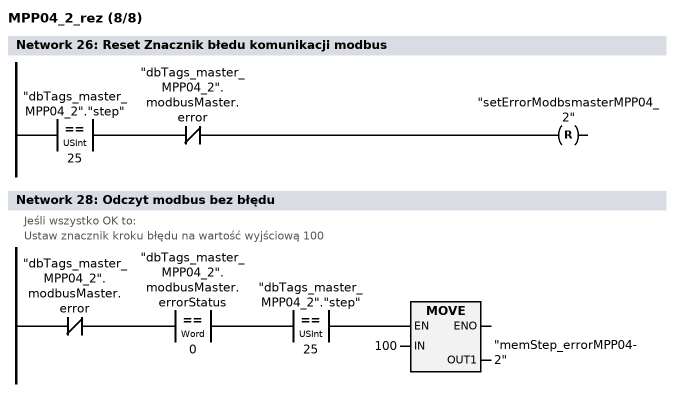
   RUNG wire#powerrail
      { S7_Templates := "SrcType := USInt" } EQ_Contact(in1 := "dbTags_master_MPP04_2"."step", in2 := 25)
      I_Contact( "dbTags_master_MPP04_2".modbusMaster.error )
      R_Coil( "setErrorModbsmasterMPP04_2" )
   END_RUNG
   // the same network as SCL:
   IF ("dbTags_master_MPP04_2"."step" = 25) AND NOT "dbTags_master_MPP04_2".modbusMaster.error THEN
       "setErrorModbsmasterMPP04_2" := FALSE;
   END_IF;
END_REGION

REGION Network 28: Odczyt modbus bez błędu
   // Jeśli wszystko OK to:
   // Ustaw znacznik kroku błędu na wartość wyjściową 100
   RUNG wire#powerrail
      I_Contact( "dbTags_master_MPP04_2".modbusMaster.error )
      { S7_Templates := "SrcType := Word" } EQ_Contact(in1 := "dbTags_master_MPP04_2".modbusMaster.errorStatus, in2 := 0)
      { S7_Templates := "SrcType := USInt" } EQ_Contact(in1 := "dbTags_master_MPP04_2"."step", in2 := 25)
      { S7_GenerateENO := "TRUE" } Move(in := 100, out1 => "memStep_errorMPP04-2")
   END_RUNG
   // the same network as SCL:
   IF NOT "dbTags_master_MPP04_2".modbusMaster.error AND ("dbTags_master_MPP04_2".modbusMaster.errorStatus = 0) AND ("dbTags_master_MPP04_2"."step" = 25) THEN
       "memStep_errorMPP04-2" := 100;
   END_IF;
END_REGION
END_FUNCTION
